FUNCTION_BLOCK EjecutarComando
VAR_INPUT
END_VAR
VAR_OUTPUT
END_VAR
VAR
	dalfa : REAL;
	dbeta : REAL;
END_VAR

IF NOT(GVL.parada) THEN 
	IF GVL.comando_actual_tipo='G00' THEN
		///inicializar regimenes a cero
		GVL.Cilindro1.regimen:=0;
		GVL.Cilindro2.regimen:=0;
		IF NOT GVL.en_objetivo_alfa THEN
	IF GVL.alfa<GVL.alfa_sp THEN
		GVL.Cilindro1.regimen:=GVL.regimen_maximo;
		ELSE IF GVL.alfa>GVL.alfa_sp THEN
		GVL.Cilindro1.regimen:=-GVL.regimen_maximo;
	END_IF
END_IF
END_IF
IF NOT GVL.en_objetivo_beta THEN
	IF GVL.beta<GVL.beta_sp THEN
		GVL.Cilindro2.regimen:=GVL.regimen_maximo;
		ELSE IF GVL.beta>GVL.beta_sp THEN
		GVL.Cilindro2.regimen:=-GVL.regimen_maximo;
	END_IF
END_IF
END_IF
	ELSE IF GVL.comando_actual_tipo='G01' THEN
		///inicializar regimenes a cero
		GVL.Cilindro1.regimen:=0;
		GVL.Cilindro2.regimen:=0;
		IF NOT GVL.en_objetivo THEN
		///determinar la diferencia con el objetivo en alfa y beta
		dalfa:=GVL.alfa_sp-GVL.alfa;
		dbeta:=GVL.beta_sp-GVL.beta;
		//si alfa está más lejos que beta
		IF ABS(dalfa)>ABS(dbeta) THEN
			IF NOT GVL.en_objetivo_alfa THEN
			IF dalfa > 0 THEN
				//mover cilindro 1 a velocidad máxima
				GVL.Cilindro1.regimen:=GVL.regimen_maximo;
				ELSE
					//o mínima
					GVL.Cilindro1.regimen:=-GVL.regimen_maximo;
				END_IF
			END_IF
				//y mover cilindro 2 a menor velocidad dbeta/dalfa
			IF NOT GVL.en_objetivo_beta THEN
				IF dbeta >0 THEN
					GVL.Cilindro2.regimen:=GVL.regimen_maximo*ABS(dbeta/dalfa);
					ELSE
						GVL.Cilindro2.regimen:=-GVL.regimen_maximo*ABS(dbeta/dalfa);
					END_IF
			END_IF

			// si beta está más lejos que alfa
			ELSE
			IF NOT GVL.en_objetivo_beta THEN
			IF dbeta > 0 THEN
				//mover cilindro 2 a velocidad máxima
				GVL.Cilindro2.regimen:=GVL.regimen_maximo;
				ELSE
					//o mínima
					GVL.Cilindro2.regimen:=-GVL.regimen_maximo;
				END_IF
			END_IF
				//y mover cilindro 1 a menor velocidad dalfa/dbeta
			IF NOT GVL.en_objetivo_alfa THEN
				IF dalfa >0 THEN
					GVL.Cilindro1.regimen:=GVL.regimen_maximo*ABS(dalfa/dbeta);
					ELSE
						GVL.Cilindro1.regimen:=-GVL.regimen_maximo*ABS(dalfa/dbeta);
					END_IF
			END_IF
			END_IF
		
		END_IF
	END_IF
	END_IF
				END_IF
	
//SI NO HE LLEGADO NO ACEPTO NUEVO COMANDO
IF NOT GVL.en_objetivo THEN
	IO.ready := FALSE;
	IO.string_out := CONCAT('Executing: ',gvl.comando_actual);
	ELSE
		IO.ready := TRUE;
		IO.string_out := concat(concat(concat(CONCAT( 'Ready at Xc=', INT_TO_STRING(IO.Xc_ADS)), 'mm, Yc='),  INT_TO_STRING(IO.Yc_ADS)) , 'mm');
END_IF

//SI EL SETPOINT ES ERRONEO, AVISAR Y ABRIR CANAL
IF GVL.error THEN
		IO.ready := TRUE;
		IO.string_out := 'Objetivo inválido, mandar nuevo comando';
END_IF

//SI EL COMANDO ES DESCONOCIDO, AVISAR Y ABRIR CANAL

IF GVL.comando_actual='Comando desconocido' THEN
			IO.ready := TRUE;
		IO.string_out := 'Comando desconocido, mandar nuevo comando';
END_IF

END_FUNCTION_BLOCK

(* stored: Version 1.1.0.1, ProductVersion 3.1.4024.4
   POU EjecutarComando: Id {44be1fb8-f127-407a-84ef-7ce9815273f2}, SpecialFunc None *)
